Staubli VAL3: CommType.dtx

public num nRequest = 2
public num nResponse = 3
